Fanuc KAREL source: kt00908.KL

PROGRAM KT00908
%STACKSIZE=65535
%PRIORITY=65535
%NOLOCKGROUP
VAR
P1 : POSITION
P2 : POSITION
OUT : VECTOR
BEGIN
OUT=ORIENT(P1)
END KT00908
